FUNCTION_BLOCK AX_ATM_FB_TP (* standard timer function block (pulse) with AX/ATM Adapter, PT and ET as adapters *)
  (* Standard: 61131-3; Classification: standard timer function block; Description: Copyright (c) 2026 HR Agrartechnik GmbH This program and the accompanying materials are made available under the terms of the Eclipse Public License 2.0 which is available at https://www.eclipse.org/legal/epl-2.0/ SPDX-License-Identifier: EPL-2.0 Wie AX_FB_TP, aber PT (Socket) und ET (Plug) sind ATM-Adapter statt einfacher Datenvariablen, s. AX_ATM_FB_TON fuer die Begruendung. *)
  (* Version 1.0, 2026-08-13, Franz Höpfinger, HR Agrartechnik GmbH, initial API and implementation *)
  PACKAGE adapter::iec61131::timers;
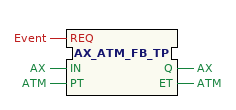
  EVENT_INPUT
    REQ; (* Normal Execution Request (non-triggering); Anwendung haengt hier periodisch einen E_CYCLE an, damit ET aktualisiert wird *)
  END_EVENT
  SOCKETS
    IN : adapter::types::unidirectional::AX; (* Input *)
    PT : adapter::types::unidirectional::ATM; (* Pulse time *)
  END_SOCKETS
  PLUGS
    Q : adapter::types::unidirectional::AX; (* Output *)
    ET : adapter::types::unidirectional::ATM; (* Elapsed time, Event nur bei Wertaenderung *)
  END_PLUGS
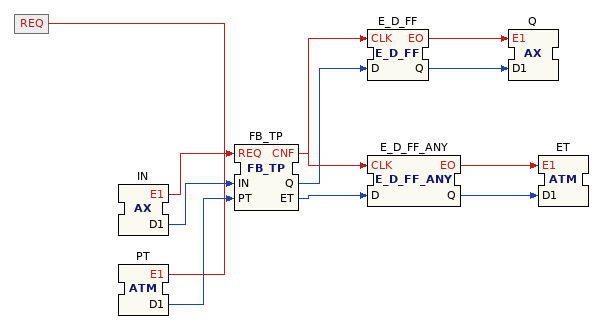
  FBS
    FB_TP : iec61131::timers::FB_TP;
    E_D_FF : iec61499::events::E_D_FF;
    E_D_FF_ANY : iec61499::events::E_D_FF_ANY;
  END_FBS
  EVENT_CONNECTIONS
    IN.E1 TO FB_TP.REQ;
    REQ TO FB_TP.REQ;
    FB_TP.CNF TO E_D_FF.CLK;
    E_D_FF.EO TO Q.E1;
    FB_TP.CNF TO E_D_FF_ANY.CLK;
    E_D_FF_ANY.EO TO ET.E1;
    PT.E1 TO FB_TP.REQ;
  END_CONNECTIONS
  DATA_CONNECTIONS
    IN.D1 TO FB_TP.IN;
    PT.D1 TO FB_TP.PT;
    FB_TP.Q TO E_D_FF.D;
    E_D_FF.Q TO Q.D1;
    FB_TP.ET TO E_D_FF_ANY.D;
    E_D_FF_ANY.Q TO ET.D1;
  END_CONNECTIONS
END_FUNCTION_BLOCK
